FUNCTION_BLOCK FB_ValveOutput
VAR_INPUT
	bEnable	: BOOL;
	bDeadBandCompOn	:BOOL;
	stValveDeadBand	: ST_ValveDeadBand;
	fNormalizedInput	: LREAL;
END_VAR
VAR_OUTPUT
	bEnableValveOutput	: BOOL;
	nOutput 			: INT;
END_VAR
VAR
	nOffset		: INT := 19660;
	nMaxValue	: INT := 29490;
	nMinValue	: INT := 9830;
	nTempOutput	: INT;
END_VAR

IF bDeadBandCompOn THEN
	IF fNormalizedInput > 0.0 THEN
		nTempOutput := LREAL_TO_INT(ABS(fNormalizedInput*(stValveDeadBand.fPosMax - stValveDeadBand.fPosMin) + stValveDeadBand.fPosMin));
	ELSIF fNormalizedInput < 0.0 THEN
		nTempOutput := LREAL_TO_INT(ABS(fNormalizedInput*(stValveDeadBand.fNegMax - stValveDeadBand.fNegMin) - stValveDeadBand.fNegMin));
	ELSE
		nTempOutput := nOffset;
	END_IF
ELSE
	IF fNormalizedInput > 0.0 THEN
		nTempOutput := LREAL_TO_INT(ABS(fNormalizedInput*(32767.0 - 19660.0) + 19660.0));
	ELSIF fNormalizedInput < 0.0 THEN
		nTempOutput := LREAL_TO_INT(ABS(fNormalizedInput*(0.0 - 19660.0) + 19660.0));
	ELSE 
		nTempOutput := nOffset;
	END_IF
END_IF

IF bEnable THEN
	nOutput := LIMIT(nMinValue, nTempOutput, nMaxValue);
	bEnableValveOutput := TRUE;
ELSE
	nOutput := nOffset;
	bEnableValveOutput := FALSE;
END_IF

END_FUNCTION_BLOCK

(* stored: Version 1.1.0.1, ProductVersion 3.1.4024.12
   POU FB_ValveOutput: Id {4043da72-f6c8-4226-b517-a0e796dc44f2}, SpecialFunc None *)
